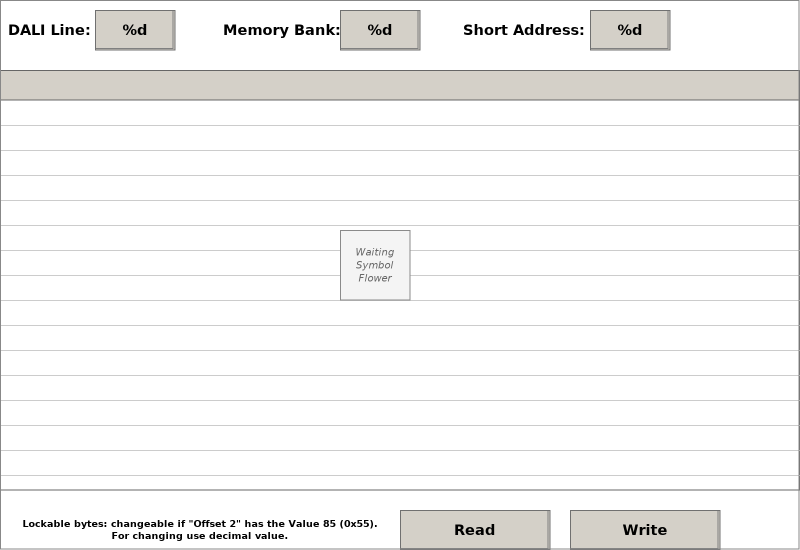
VISUALIZATION Visu_Part103MemoryBank  // 800x550
    Table (0,70 800x420), data array: DALI_Commissioning.fbPart103MemoryPages.aMemoryBank
        p3854506369: DALI_Commissioning.fbPart103MemoryPages.aMemoryBank[INDEX].sOffset
        p1892666644: DALI_Commissioning.fbPart103MemoryPages.aMemoryBank[INDEX].sName
        p338671338: DALI_Commissioning.fbPart103MemoryPages.aMemoryBank[INDEX].nValueDec
        p2170511999: DALI_Commissioning.fbPart103MemoryPages.aMemoryBank[INDEX].nValueHex
        p1755163831: Value Dec
        p4092479075: Value Hex
        p1137915858: DALI_Commissioning.fbPart103MemoryPages.nOffset
        Columns.Column.[2].Template: DALI_Commissioning.fbPart103MemoryPages.aNoValue[INDEX]; DALI_Commissioning.fbPart103MemoryPages.nMemoryBank=0; OnMouseClick: write the text variable via Default, min 0, max 255, title "Lockable variable decimal"
        Columns.Column.[0].Template: DALI_Commissioning.fbPart103MemoryPages.aNoValue[INDEX]
        Columns.Column.[1].Template: DALI_Commissioning.fbPart103MemoryPages.aNoValue[INDEX]
        Columns.Column.[3].Template: DALI_Commissioning.fbPart103MemoryPages.aNoValue[INDEX]; OnMouseClick: write the text variable via Default, title "Lockable variable hexadecimal"
    Button (400,510 150x40), "Read"
        OnMouseClick: execute { DALI_Commissioning.fbPart103MemoryPages.bRead := TRUE; }
    Button (570,510 150x40), "Write"
        OnMouseClick: execute { DALI_Commissioning.fbPart103MemoryPages.bWrite := TRUE; }
    Textfield (15,510 370x40), "Lockable bytes: changeable if "Offset 2" has the Value 85 (0x55). For changing use decimal value."
    WaitingSymbolFlower (340,230 70x70), invisible if: DALI_Commissioning.fbPart103MemoryPages.bHideWaitSymbol
    Textfield (460,10 130x40), "Short Address:"
    Button (590,10 80x40), "%d", text variable: DALI_Commissioning.fbPart103MemoryPages.nAddress
        OnMouseClick: write the text variable via Default, min 0, max 63, title "Insert Short Address"
    Group (220,10 200x40)
        Textfield (0,0 150x40), "Memory Bank:"
        Button (120,0 80x40), "%d", text variable: DALI_Commissioning.fbPart103MemoryPages.nMemoryBank
            OnMouseClick: write the text variable via Default, min 0, max 255, title "Insert Memory Bank"
    Group (5,10 170x40)
        Textfield (0,0 110x40), "DALI Line:"
        Button (90,0 80x40), "%d", text variable: GVL_Internal.nDALILine
            OnMouseClick: write the text variable via Default, min 1, max 10, title "Choose line"
END_VISUALIZATION

(* stored: Version 1.1.0.1, ProductVersion 3.1.4024.9
   Visu Visu_Part103MemoryBank: Id {eed2b28d-80eb-490f-b9fc-9f1cee153391} *)
